Fanuc KAREL source: ko00043.KL

-- PROVISIONAL review KL for V770-1; original PC SHA256 a58774b8d90b91fb305458081975adecc120e827e6e939358759616ec84f773d
-- Incomplete behavior may be omitted. Consult companion uncertainty JSON. Do not deploy.
PROGRAM KO00043
%NOLOCKGROUP
BEGIN
  -- UNRESOLVED_PC offsets 5-12; opcodes 9D,23
  -- UNRESOLVED_PC offsets 17-69; opcodes 27,27,49,7E,AD,27,49,7E,AD,22,31,7E,4A
  -- UNRESOLVED_PC offsets 74-78; opcodes 7F
END KO00043
